// Mitsubishi GX Works2 project: 0624(자기유지회로)   PLC: Q02/Q02H

PROGRAM MAIN
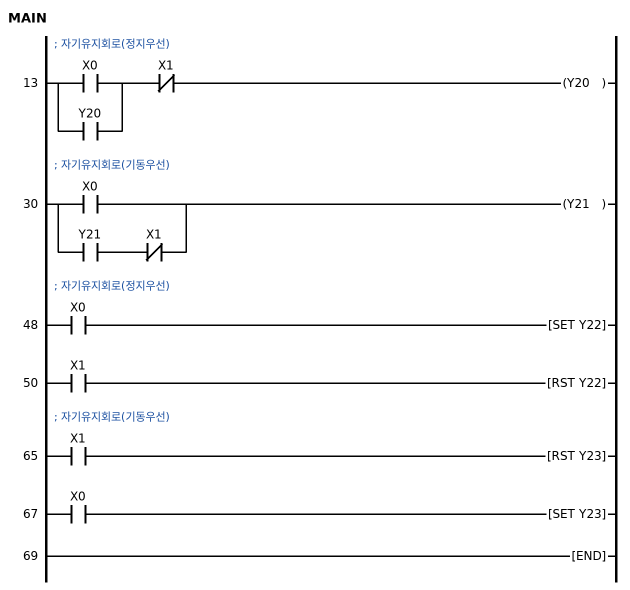
; 자기유지회로(정지우선)
13    LD      X0
      OR      Y20
      ANI     X1
      OUT     Y20
; 자기유지회로(기동우선)
30    LD      X0
      LD      Y21
      ANI     X1
      ORB
      OUT     Y21
; 자기유지회로(정지우선)
48    LD      X0
      SET     Y22
50    LD      X1
      RST     Y22
; 자기유지회로(기동우선)
65    LD      X1
      RST     Y23
67    LD      X0
      SET     Y23
69    END
END_PROGRAM
